INTERFACE ITFComponent EXTENDS __System.IQueryInterface

/// Get's or set's a value indicating whether this component is active or not.
PROPERTY Active : BOOL
GET
END_GET
SET
END_SET
END_PROPERTY

/// Get's value representing the component state.
PROPERTY ClearText : WSTRING(255)
GET
END_GET
END_PROPERTY

PROPERTY ID : INT
GET
END_GET
SET
END_SET
END_PROPERTY

/// Get's value representing the component state.
PROPERTY LastError : T_MaxString
GET
END_GET
END_PROPERTY

PROPERTY Logger : I_Logger
SET
END_SET
END_PROPERTY

PROPERTY Name : ST_Text
GET
END_GET
SET
END_SET
END_PROPERTY

PROPERTY ObjectId : WSTRING
GET
END_GET
END_PROPERTY

PROPERTY Path : String
GET
END_GET
END_PROPERTY

PROPERTY RefsValid : BOOL
GET
END_GET
END_PROPERTY

/// Reset component logic
{attribute 'object_name' := 'Reset'}
METHOD Reset
END_METHOD

/// Run component logic
{attribute 'object_name' := 'Run'}
METHOD Run : E_ComponentState
END_METHOD

/// Get's value representing the component state.
PROPERTY State : E_ComponentState
GET
END_GET
END_PROPERTY

/// Get's value representing the component state.
PROPERTY StateToString : STRING
GET
END_GET
END_PROPERTY

PROPERTY Typ : E_ComponentType
GET
END_GET
END_PROPERTY

END_INTERFACE

(* stored: Version 1.1.0.1, ProductVersion 3.1.4024.11
   Itf ITFComponent: Id {0c339870-3919-4156-9e10-4458967cc3e3}
   Property Active: Id {a4013bac-f678-40d6-b6e3-75f80b396d7b}
   Get Get: Id {af35816a-6e99-4110-b78f-ac05c3ac3868}
   Set Set: Id {79941203-7a00-4cd8-82bc-f02302f41a88}
   Property ClearText: Id {1b270129-2b79-4ed2-8681-18554c509971}
   Get Get: Id {6beec932-c0ca-48e0-91e5-86775b94b797}
   Property ID: Id {d6eb581a-9300-43d2-a537-fd27c418df38}
   Get Get: Id {a70e8b71-2e06-4591-a3d1-6a2521787bc6}
   Set Set: Id {0397acb8-1194-48f7-a076-a7b502c58cc9}
   Property LastError: Id {f1d9d119-6784-4c74-950f-734bdedcbab4}
   Get Get: Id {882a1694-bf62-497a-8196-c43862a41266}
   Property Logger: Id {c94da13d-936f-4604-8f56-f9d4637d5aa0}
   Set Set: Id {86accb3c-15ac-4d20-b299-f862adcd0a23}
   Property Name: Id {dfe3cfb1-960f-481b-9895-7c3d2fdb66bb}
   Get Get: Id {3ed505ba-48a7-4459-a5b0-60e9cc302605}
   Set Set: Id {4fd43b83-a34d-4197-ae89-db48925894aa}
   Property ObjectId: Id {3b25599c-30b5-4fd6-958e-979f9ea8eddb}
   Get Get: Id {05c23f4f-324e-4902-a8e9-ff8c3e111e4e}
   Property Path: Id {d49383b0-7900-4755-8881-e6510a11411d}
   Get Get: Id {81f6854d-d864-4189-ad35-0ff1836e1149}
   Property RefsValid: Id {fa04309d-9f80-475c-97db-b5a91f3a4fc4}
   Get Get: Id {be8fe2db-8038-4f53-acbc-4f79a5540e2b}
   Method Reset: Id {d20f6564-ac00-4f07-b6e7-4efc746c414a}
   Method Run: Id {9456d1b6-8b95-48fd-bbab-7ac1c5ad6db3}
   Property State: Id {62ee10f7-b429-4216-b697-b5f173ac2511}
   Get Get: Id {55b5c8bf-e40a-4d54-a4c5-8ddf14ed0583}
   Property StateToString: Id {6b6e811f-0f6a-45c4-af3a-a9178954bbe3}
   Get Get: Id {8b6e04fc-9441-4459-b058-ef6def792db0}
   Property Typ: Id {600151d1-2b3c-4c87-a5bb-ed8db31b21c9}
   Get Get: Id {a79651d5-3615-41ad-8b6b-c03c92d545e8} *)
